(* IEC 61131-3 sources: GitHub_Test/YF_DoubleAGV/CVC_TcpTest/PLC (part 2) *)

   END_STRUCT;
END_TYPE
TYPE
    SSIO_T :
    STRUCT
        LogicalLine : DINT ;   (* Logical SSIO line.  *)
        UnitNumber : DINT ;   (* Unit id in a logical line.  *)
        InputOutputID : DINT ;   (* ID of input/output in unit.  *)
        RequestType : DINT ;   (* 0:Read input status, 1:Read output status, 2:Set output status.  *)
        SetStatus : DINT ;   (* The status to set in case of a Set output status request, 0:OFF, 1:ON, 2:Flash 1Hz.  *)
        Status : DINT ;   (* The returned status in case of a read request. Valid only when SSIO_ENO is set.  *)
        SSIO_EN : BOOL ;   (* First set SSIO address and request type then set this property to initiate a SSIO request. Clear when SSIO_ENO is set and Status has been read.  *)
        SSIO_ENO : BOOL ;   (* Set by background software when the SSIO request has been executed. For a read request this means that the reply can be read from the Status property.  *)
        Error : DINT ;   (* 0:No error, 1:Timeout.  *)

   END_STRUCT;
END_TYPE
TYPE
    CanOpenMaster_T :
    STRUCT
        MasterExecutionPeriod : DINT ;   (* Execution period for the CANopen master component. Unit is [ms].  *)
        SyncPeriod : DINT ;   (* Sync producer period given in multiples of MasterExecutionPeriod.  *)
        CollectTimeout : DINT ;   (* Collect timeout before can server enters safe state  *)
        CanMasterCmd : DINT ;   (* Command to CAN master when CanMasterEN is set, 1 = RestartCan, 2 = GoToSafeState  *)
        CanMasterCmdEN : BOOL ;   (* Commands CAN master to CanMasterCmd. Clear it when CanMasterCmdENO is set.  *)
        CanMasterCmdENO : BOOL ;   (* Set by background when commands CAN master to CanMasterCmd. Cleared when CanMasterEN is cleared.  *)
        NMTState : UDINT ;   (* The current CANopen state of the vehicle controller. Interpretation:
                        Initializing (0) = loading definition,
                        Stopped (4) = unable to start due to fatal definition error,
                        Operational (5) = The vehicle controller fully operational either in normal state or in safestate,
                        PreOperational (127) = pre-operational, configuration of slave devices,
                        Unknown (255) = state undefined, no communication with node  *)
        State : DINT ;   (* Current state of the CanOpenMaster application, 0 = NormalState, 1 = SafeState. When any error is detected that PLC does not handle, the vehicle controller will enter SafeState. Information about the error causing SafeState is available in properties StatusText, EMCY_NodeID, EMCY_Code, EMCY_ErrReg, EMCY_Byte1, etc. SafeState is a passive/diagnostic state and AllOk will be set to false.  *)
        StatusText : STRING ;   (* Text description of error that caused the vehicle controller to enter SafeState. Only valid when State = SafeState.  *)
        EMCY_BusID : DINT ;   (* Bus ID that reported the error. Only valid when State = SafeState.  *)
        EMCY_NodeID : DINT ;   (* Node ID that reported the error. Only valid when State = SafeState.  *)
        EMCY_Code : DINT ;   (* CANopen emergency code, see device documentation. Only valid when State = SafeState.  *)
        EMCY_ErrReg : DINT ;   (* Error registry. Only valid when State = SafeState.  *)
        EMCY_Byte1 : DINT ;   (* Manufacturer specific field, byte 1. Only valid when State = SafeState.  *)
        EMCY_Byte2 : DINT ;   (* Manufacturer specific field, byte 2. Only valid when State = SafeState.  *)
        EMCY_Byte3 : DINT ;   (* Manufacturer specific field, byte 3. Only valid when State = SafeState.  *)
        EMCY_Byte4 : DINT ;   (* Manufacturer specific field, byte 4. Only valid when State = SafeState.  *)
        EMCY_Byte5 : DINT ;   (* Manufacturer specific field, byte 5. Only valid when State = SafeState.  *)

   END_STRUCT;
END_TYPE
TYPE
    CanOpenEmergency_T :
    STRUCT
        EmcyEN : BOOL ;   (* Set by background when emergency data is available for a CAN device that has FailureAction set to PLC. Cleared when ENO is set.  *)
        EmcyENO : BOOL ;   (* Set by PLC when read emergency data, cleared when EN is cleared.  *)
        BusID : DINT ;   (* CAN bus id.  *)
        NodeID : DINT ;   (* CAN node id.  *)
        Code : DINT ;   (* Error code according to CANopen standard. When an emergency is generated by background program (node id is negative), the node id for the node it concerns is the last 5 bits of the code.  *)
        ErrReg : DINT ;   (* Error register according to CANopen standard.  *)
        Byte1 : DINT ;   (* Manufacturer specific error field according to CANopen standard.  *)
        Byte2 : DINT ;   (* Manufacturer specific error field according to CANopen standard.  *)
        Byte3 : DINT ;   (* Manufacturer specific error field according to CANopen standard.  *)
        Byte4 : DINT ;   (* Manufacturer specific error field according to CANopen standard.  *)
        Byte5 : DINT ;   (* Manufacturer specific error field according to CANopen standard.  *)

   END_STRUCT;
END_TYPE
TYPE
    PLCEmergency_T :
    STRUCT
        Canbus : DINT ;   (* Bus to send emergency on. 0 = first bus, 1 = second bus.  *)
        Code : DINT ;   (* Error code according to CANopen standard.  *)
        ErrReg : DINT ;   (* Error register according to CANopen standard.  *)
        Byte1 : DINT ;   (* Manufacturer specific error field according to CANopen standard.  *)
        Byte2 : DINT ;   (* Manufacturer specific error field according to CANopen standard.  *)
        Byte3 : DINT ;   (* Manufacturer specific error field according to CANopen standard.  *)
        Byte4 : DINT ;   (* Manufacturer specific error field according to CANopen standard.  *)
        Byte5 : DINT ;   (* Manufacturer specific error field according to CANopen standard.  *)
        EmcyEN : BOOL ;   (* Set by PLC when emergency data is available. Cleared by PLC when ENO is set.  *)
        EmcyENO : BOOL ;   (* Set by the vehicle controller when emergency data has been read. Cleared by the vehicle controller when EN is cleared.  *)

   END_STRUCT;
END_TYPE
TYPE
    SlavebusControl_T :
    STRUCT
        EnterPreOpEN : BOOL ;   (* Set by background when requesting to enter NMT state pre-operational. Cleared when ENO is set.  *)
        EnterPreOpENO : BOOL ;   (* Set by PLC when transition to NMT state pre-operational is granted. Cleared when EN is cleared.  *)

   END_STRUCT;
END_TYPE
TYPE
    PPA_T :
    STRUCT
        LaserScannerRef : STRING ;   (* Reference to the Laser scanner component  *)
        FrontWheelRef : STRING ;   (* Reference to the front wheel component  *)
        SteerEncRef : STRING ;   (* Symbol address where the steer encoder offset is defined. Ex: SDIO_1.SteerEncOffset  *)
        CurrentState : DINT ;   (* Current or last state of action:
0 = Idle
1 = Driving sequence 1
2 = Driving sequence 2
3 = Driving sequence 3
4 = Driving sequence 4
5 = Driving sequence 5
6 = Estimation in progress
7 = Estimation done result ok  *)
        EstimationProgress : DINT ;   (* Progressbar during calculation  *)
        CmdID : DINT ;   (* ID of current movement 1-5  *)
        ErrorID : DINT ;   (* Error Id for error condition. 0 = no error  *)
        CmdDone : DINT ;   (* Indicates completion of requested command.  *)
        SteerEncOffset : DINT ;   (* Calculated value  *)
        LaserScannerX : DINT ;   (* Calculated value  *)
        LaserScannerY : DINT ;   (* Calculated value  *)
        LaserScannerAngle : REAL ;   (* Calculated value  *)

   END_STRUCT;
END_TYPE
TYPE
    LanSerialPort_T :
    STRUCT
        Protocol : DINT ;   (* Protocol used for IP communication.  *)
        IP : STRING ;   (* In case of Protocol set to UDP client or TCP client this should be set
to the IP address of the UDP/TCP server that the PLC connects to. With
Protocol set to UDP server or TCP server this specify the IP address of
the vehicle controller which clients should use.

In the case of Protocol set to UDP server or TCP server, the special
value "LAN" means that connections are only allowed on the
LAN interface and the special value "ANY" allows connections
on both the LAN interface and the WLAN interface.

Changing the address from the PLC will result in the connection being
closed. The new IP address will be used in the next PLC loop serial
read/write.  Note! It is not possible to change the address for a
range sensor connected using a LAN-serial-adapter.  *)
        Port : DINT ;   (* In case of Protocol set to UDP client or TCP client this should be set
to the port of the UDP/TCP server that the PLC connects to. With
Protocol set to UDP server or TCP server this specify the port on the
vehicle controller that the PLC opens for connections.

Changing the port from the PLC will result in the connection being
closed. The new port will be used in the next PLC loop serial
read/write.  Note! It is not possible to change the port for a range
sensor connected using a LAN-serial-adapter.  *)
        SendBuffer : BOOL ;   (* With SendBuffer set, outgoing data is sent over IP when the PLC
function block NDC_SERIAL_WRITE is called with argument
LENGTH=0. Without SendBuffer set, data is sent immediately but each IP
packet will contain at most 32 bytes data with more IP traffic as a
result.  *)

   END_STRUCT;
END_TYPE
TYPE
    UserDefined_T :
    STRUCT
        HeartBeatTimeOut : BOOL ;   (*   *)
        MasterErrorStop : BOOL ;   (*   *)
        Boolean_3 : BOOL ;   (*   *)
        Boolean_4 : BOOL ;   (*   *)
        Boolean_5 : BOOL ;   (*   *)
        Boolean_6 : BOOL ;   (*   *)
        Boolean_7 : BOOL ;   (*   *)
        Boolean_8 : BOOL ;   (*   *)
        Boolean_9 : BOOL ;   (*   *)
        Boolean_10 : BOOL ;   (*   *)
        Boolean_11 : BOOL ;   (*   *)
        Boolean_12 : BOOL ;   (*   *)
        Boolean_13 : BOOL ;   (*   *)
        Boolean_14 : BOOL ;   (*   *)
        Boolean_15 : BOOL ;   (*   *)
        Boolean_16 : BOOL ;   (*   *)
        Boolean_17 : BOOL ;   (*   *)
        Boolean_18 : BOOL ;   (*   *)
        Boolean_19 : BOOL ;   (*   *)
        Boolean_20 : BOOL ;   (*   *)
        Boolean_21 : BOOL ;   (*   *)
        Boolean_22 : BOOL ;   (*   *)
        Boolean_23 : BOOL ;   (*   *)
        Boolean_24 : BOOL ;   (*   *)
        Boolean_25 : BOOL ;   (*   *)
        Boolean_26 : BOOL ;   (*   *)
        Boolean_27 : BOOL ;   (*   *)
        Boolean_28 : BOOL ;   (*   *)
        Boolean_29 : BOOL ;   (*   *)
        Boolean_30 : BOOL ;   (*   *)
        Integer32_1 : DINT ;   (*   *)
        Integer32_2 : DINT ;   (*   *)
        Integer32_3 : DINT ;   (*   *)
        Integer32_4 : DINT ;   (*   *)
        Integer32_5 : DINT ;   (*   *)
        Integer32_6 : DINT ;   (*   *)
        Integer32_7 : DINT ;   (*   *)
        Integer32_8 : DINT ;   (*   *)
        Integer32_9 : DINT ;   (*   *)
        Integer32_10 : DINT ;   (*   *)
        Integer32_11 : DINT ;   (*   *)
        Integer32_12 : DINT ;   (*   *)
        Integer32_13 : DINT ;   (*   *)
        Integer32_14 : DINT ;   (*   *)
        Integer32_15 : DINT ;   (*   *)
        Integer32_16 : DINT ;   (*   *)
        Integer32_17 : DINT ;   (*   *)
        Integer32_18 : DINT ;   (*   *)
        Integer32_19 : DINT ;   (*   *)
        Integer32_20 : DINT ;   (*   *)
        Integer32_21 : DINT ;   (*   *)
        TractionEncSpeed : DINT ;   (*   *)
        TractionSetSpeed : DINT ;   (*   *)
        FrontSetSpeed : DINT ;   (*   *)
        FrontEncSpeed : DINT ;   (*   *)
        FrontSetAngle : DINT ;   (*   *)
        FrontEncAngle : DINT ;   (*   *)
        RearSetSpeed : DINT ;   (*   *)
        RearEncSpeed : DINT ;   (*   *)
        RearSetAngle : DINT ;   (*   *)
        RearEncAngle : DINT ;   (*   *)
        VirFrontSetSpeed : DINT ;   (*   *)
        VirFrontEncSpeed : DINT ;   (*   *)
        VirFrontSetAngle : DINT ;   (*   *)
        VirFrontEncAngle : DINT ;   (*   *)
        VirRearSetSpeed : DINT ;   (*   *)
        VirRearEncSpeed : DINT ;   (*   *)
        VirRearSetAngle : DINT ;   (*   *)
        VirRearEncAngle : DINT ;   (*   *)
        Integer32_40 : DINT ;   (*   *)
        VirFFeedbackSpeed : DINT ;   (*   *)
        VirFFeedbackAngle : DINT ;   (*   *)
        VirRFeedbackSpeed : DINT ;   (*   *)
        VirRFeedbackAngle : DINT ;   (*   *)
        Integer32_45 : DINT ;   (*   *)
        Integer32_46 : DINT ;   (*   *)
        Integer32_47 : DINT ;   (*   *)
        Integer32_48 : DINT ;   (*   *)
        Integer32_49 : DINT ;   (*   *)
        Integer32_50 : DINT ;   (*   *)
        Integer32_51 : DINT ;   (*   *)
        Integer32_52 : DINT ;   (*   *)
        Integer32_53 : DINT ;   (*   *)
        Integer32_54 : DINT ;   (*   *)
        Integer32_55 : DINT ;   (*   *)
        Integer32_56 : DINT ;   (*   *)
        Integer32_57 : DINT ;   (*   *)
        Integer32_58 : DINT ;   (*   *)
        Integer32_59 : DINT ;   (*   *)
        Integer32_60 : DINT ;   (*   *)

   END_STRUCT;
END_TYPE
TYPE
    SDIO_T :
    STRUCT
        SteerRegP : UINT ;   (* Steering Regulator P Gain  *)
        SteerRegI : UINT ;   (* Steering Regulator I Gain  *)
        SteerRegILimit : UINT ;   (* Steering Regulator I Gain Limit  *)
        SteerRegD : UINT ;   (* Steering Regulator D Gain  *)
        SteerRegPIDLimit : UINT ;   (* Limits the effect of feedback on the steering regulator.
The unit is mV in an SDIO-FSA system.
For system only feeding the regulator output on the canbus, the value is pure binary.  *)
        SteerRegOutOffset : INT ;   (* Output offset for the steering regulator.
This offset is added to the regulator output after the PID regulation.
The unit is mV in an SDIO-FSA system.
For system only feeding the regulator output on the canbus, the value is pure binary.  *)
        SteerRegOutLimit : UINT ;   (* Total output limit of the steering regulator.
The unit is mV in an SDIO-FSA system.
For system only feeding the regulator output on the canbus, the value is pure binary.  *)
        SteerRegFailureDelay : UINT ;   (* Delay before safe state in absence of correct feedback movement  *)
        SteerRegCheckOutHysteres : UINT ;   (* Feedback movement is checked when the regulator output is larger than this level  *)
        SteerEncScale : UINT ;   (* Steering Encoder Scale  *)
        SteerEncOffset : INT ;   (* Steering Encoder Offset (Position of Sync pulse)  *)
        SteerEncSyncFilter : UINT ;   (* Steering Encoder Sync Filter Window, unit [pulses]. Filter is applied with half of the value to the right and half of the value to the left of the last valid sync pulse. 0 = Filter disabled. OBS! Disabling the sync filter can be a serious safety issue!  *)
        SteerEncSyncEmergency : BOOL ;   (* Steering Encoder Sync Emergency. 0 = Sync Emergency disabled. OBS! Disabling the sync emergency can be a serious safety issue!  *)
        SteerEncSyncEnable : BOOL ;   (* Enable signal for encoder sync mechanism. Usually needed when having a multiturning steering encoder  *)
        SyncGateInput : USINT ;   (* Digital input used for sync gate. 0 = disabled  *)
        DriveRegFeedForward : UINT ;   (* Driving Regulator FeedForward Gain  *)
        DriveRegOffset : UINT ;   (* Driving Regulator Offset  *)
        DriveRegP : UINT ;   (* Driving Regulator P Gain  *)
        DriveRegI : UINT ;   (* Driving Regulator I Gain  *)
        DriveRegILimit : UINT ;   (* Driving Regulator I Gain Limit  *)
        DriveRegD : UINT ;   (* Driving Regulator D Gain  *)
        DriveRegPIDLimit : UINT ;   (* Limits the effect of feedback on the drive regulator.
The unit is mV in an SDIO-FSA system.
For system only feeding the regulator output on the canbus, the value is pure binary.  *)
        DriveRegOutOffset : INT ;   (* Output offset for the drive regulator.
This offset is added to the regulator output after the PID regulation.
The unit is mV in an SDIO-FSA system.
For system only feeding the regulator output on the canbus, the value is pure binary.  *)
        DriveRegOutLimit : UINT ;   (* Total output limit of the drive regulator.
The unit is mV in an SDIO-FSA system.
For system only feeding the regulator output on the canbus, the value is pure binary.  *)
        DriveRegFailureDelay : UINT ;   (* Delay before safe state in absence of correct feedback movement  *)
        DriveRegCheckOutHysteres : UINT ;   (* Feedback movement is checked when the regulator output is larger than this level  *)
        DriveEncScale : UINT ;   (* Driving Encoder Scale  *)
        DigitalInput6_Polarity : BOOL ;   (* Digital Input 6 Polarity, pin #A21  *)
        FSA1Failure_Polarity : BOOL ;   (* FSA 1 Failure Polarity, pin #A20  *)
        FSA2Failure_Polarity : BOOL ;   (* FSA 2 Failure Polarity, pin #A19  *)
        DigitalInput9_Polarity : BOOL ;   (* Digital Input 9 Polarity, pin #B22  *)
        DigitalInput10_Polarity : BOOL ;   (* Digital Input 10 Polarity, pin #B23  *)
        DigitalInput11_Polarity : BOOL ;   (* Digital Input 11 Polarity, pin #A18  *)
        DigitalInput12_Polarity : BOOL ;   (* Digital Input 12 Polarity, pin #A17  *)
        DigitalOutput2_Polarity : BOOL ;   (* Digital Output 2 Polarity, pin #B7  *)
        DigitalOutput3_Polarity : BOOL ;   (* Digital Output 3 Polarity, pin #B6  *)
        DigitalOutput4_Polarity : BOOL ;   (* Digital Output 4 Polarity, pin #B5  *)
        DigitalOutput5_Polarity : BOOL ;   (* Digital Output 5 Polarity, pin #B4  *)
        DigitalOutput6_Polarity : BOOL ;   (* Digital Output 6 Polarity, pin #B1  *)
        DigitalOutput12_Polarity : BOOL ;   (* Digital Output 12 Polarity, pin #A3  *)
        AnInp1_Scale : DINT ;   (* Analog Input 1 Scale, pin #B15  *)
        AnInp2_Scale : DINT ;   (* Analog Input 2 Scale, pin #B17  *)
        AnInp3_Scale : DINT ;   (* Analog Input 3 Scale, pin #B10  *)
        AnInp4_Scale : DINT ;   (* Analog Input 4 Scale, pin #B18  *)
        AnInp5_Scale : DINT ;   (* Analog Input 5 Scale, pin #B11  *)
        AnInp6_Scale : DINT ;   (* Analog Input 6 Scale, pin #B19  *)
        AnInp7_Scale : DINT ;   (* Analog Input 7 Scale, pin #B12  *)
        AnInp8_Scale : DINT ;   (* Analog Input 8 Scale, pin #B20  *)
        AnInp9_Scale : DINT ;   (* Analog Input 9 Scale, pin #B13  *)
        AnInp10_Scale : DINT ;   (* Analog Input 10 Scale, pin #B21  *)
        AnInp11_Scale : DINT ;   (* Analog Input 11 Scale, pin #B14  *)
        AnInp1_Delta : UDINT ;   (* Asynchroneous transmission will be triggered if input has changed more than this value since last transmission.  *)
        AnInp2_Delta : UDINT ;   (* Asynchroneous transmission will be triggered if input has changed more than this value since last transmission.  *)
        AnInp3_Delta : UDINT ;   (* Asynchroneous transmission will be triggered if input has changed more than this value since last transmission.  *)
        AnInp4_Delta : UDINT ;   (* Asynchroneous transmission will be triggered if input has changed more than this value since last transmission.  *)
        AnInp5_Delta : UDINT ;   (* Asynchroneous transmission will be triggered if input has changed more than this value since last transmission.  *)
        AnInp6_Delta : UDINT ;   (* Asynchroneous transmission will be triggered if input has changed more than this value since last transmission.  *)
        AnInp7_Delta : UDINT ;   (* Asynchroneous transmission will be triggered if input has changed more than this value since last transmission.  *)
        AnInp8_Delta : UDINT ;   (* Asynchroneous transmission will be triggered if input has changed more than this value since last transmission.  *)
        AnInp9_Delta : UDINT ;   (* Asynchroneous transmission will be triggered if input has changed more than this value since last transmission.  *)
        AnInp10_Delta : UDINT ;   (* Asynchroneous transmission will be triggered if input has changed more than this value since last transmission.  *)
        AnInp11_Delta : UDINT ;   (* Asynchroneous transmission will be triggered if input has changed more than this value since last transmission.  *)
        AnInp1_Offset : DINT ;   (* Analog Input 1 Offset, pin #B15  *)
        AnInp2_Offset : DINT ;   (* Analog Input 2 Offset, pin #B17  *)
        AnInp3_Offset : DINT ;   (* Analog Input 3 Offset, pin #B10  *)
        AnInp4_Offset : DINT ;   (* Analog Input 4 Offset, pin #B18  *)
        AnInp5_Offset : DINT ;   (* Analog Input 5 Offset, pin #B11  *)
        AnInp6_Offset : DINT ;   (* Analog Input 6 Offset, pin #B19  *)
        AnInp7_Offset : DINT ;   (* Analog Input 7 Offset, pin #B12  *)
        AnInp8_Offset : DINT ;   (* Analog Input 8 Offset, pin #B20  *)
        AnInp9_Offset : DINT ;   (* Analog Input 9 Offset, pin #B13  *)
        AnInp10_Offset : DINT ;   (* Analog Input 10 Offset, pin #B21  *)
        AnInp11_Offset : DINT ;   (* Analog Input 11 Offset, pin #B14  *)
        Enc1AngularSpeed : INT ;   (* Encoder 1 Angular Speed  *)
        Enc1Angle : INT ;   (* Encoder 1 Angle  *)
        Enc1SyncValid : BOOL ;   (* Encoder 1 Sync Valid  *)
        Enc1Warning : BOOL ;   (* Encoder 1 Warning  *)
        Enc2Dist : UINT ;   (* Encoder 2 Distance  *)
        Enc2Speed : INT ;   (* Encoder 2 Speed  *)
        SetAngle : INT ;   (* Set Angle  *)
        SteerEnable : BOOL ;   (* Steering Control Enable  *)
        SetSpeed : INT ;   (* Set Speed  *)
        DriveEnable : BOOL ;   (* Driving Control Enable  *)
        Reserved_DigitalInput1 : BOOL ;   (* Reserved Digital Input 1 (Enc 1 A, pin #A14)  *)
        Reserved_DigitalInput2 : BOOL ;   (* Reserved Digital Input 2 (Enc 1 B, pin #A22)  *)
        Reserved_DigitalInput3 : BOOL ;   (* Reserved Digital Input 3 (Enc 1 Sync, pin #A7)  *)
        Reserved_DigitalInput4 : BOOL ;   (* Reserved Digital Input 4 (Enc 2 A, pin #A6)  *)
        Reserved_DigitalInput5 : BOOL ;   (* Reserved Digital Input 5 (Enc 2 B, pin #A13)  *)
        DigitalInput6 : BOOL ;   (* Digital Input 6 value, pin #A21  *)
        FSA1Failure : BOOL ;   (* FSA 1 Failure value, pin #A20  *)
        FSA2Failure : BOOL ;   (* FSA 2 Failure value, pin #A19  *)
        DigitalInput9 : BOOL ;   (* Digital Input 9 value, pin #B22  *)
        DigitalInput10 : BOOL ;   (* Digital Input 10 value, pin #B23  *)
        DigitalInput11 : BOOL ;   (* Digital Input 11 value, pin #A18  *)
        DigitalInput12 : BOOL ;   (* Digital Input 12 value, pin #A17  *)
        AllOK_DigitalOutput1 : BOOL ;   (* Reserved Digital Output 1 (All-OK, pin #B8)  *)
        DigitalOutput2 : BOOL ;   (* Digital Output 2 value, pin #B7  *)
        DigitalOutput3 : BOOL ;   (* Digital Output 3 value, pin #B6  *)
        DigitalOutput4 : BOOL ;   (* Digital Output 4 value, pin #B5  *)
        DigitalOutput5 : BOOL ;   (* Digital Output 5 value, pin #B4  *)
        DigitalOutput6 : BOOL ;   (* Digital Output 6 value, pin #B1  *)
        DigitalOutput12 : BOOL ;   (* Digital Output 12 value, pin #A3  *)
        AnalogInput1 : INT ;   (* Analog Input 1 value, pin #B15. The value is the applied input voltage (in Volts) * Scale + Offset  *)
        AnalogInput2 : INT ;   (* Analog Input 2 value, pin #B17. The value is the applied input voltage (in Volts) * Scale + Offset  *)
        AnalogInput3 : INT ;   (* Analog Input 3 value, pin #B10. The value is the applied input voltage (in Volts) * Scale + Offset  *)
        AnalogInput4 : INT ;   (* Analog Input 4 value, pin #B18. The value is the applied input voltage (in Volts) * Scale + Offset  *)
        AnalogInput5 : INT ;   (* Analog Input 5 value, pin #B11. The value is the applied input voltage (in Volts) * Scale + Offset  *)
        AnalogInput6 : INT ;   (* Analog Input 6 value, pin #B19. The value is the applied input voltage (in Volts) * Scale + Offset  *)
        AnalogInput7 : INT ;   (* Analog Input 7 value, pin #B12. The value is the applied input voltage (in Volts) * Scale + Offset  *)
        AnalogInput8 : INT ;   (* Analog Input 8 value, pin #B20. The value is the applied input voltage (in Volts) * Scale + Offset  *)
        AnalogInput9 : INT ;   (* Analog Input 9 value, pin #B13. The value is the applied input voltage (in Volts) * Scale + Offset  *)
        AnalogInput10 : INT ;   (* Analog Input 10 value, pin #B21. The value is the applied input voltage (in Volts) * Scale + Offset  *)
        AnalogInput11 : INT ;   (* Analog Input 11 value, pin #B14. The value is the applied input voltage (in Volts) * Scale + Offset  *)
        PWMOutput1 : INT ;   (* PWM Output 1 value, pin #A5. The value is the duty cycle of the output.  *)
        PWMOutput2 : INT ;   (* PWM Output 2 value, pin #A12. The value is the duty cycle of the output.  *)
        PWMOutput3 : INT ;   (* PWM Output 3 value, pin #A11. The value is the duty cycle of the output.  *)
        Reg1Output : INT ;   (* Regulator 1 output value  *)
        Reg2Output : INT ;   (* Regulator 2 output value  *)
        GroundFaultEvent : BOOL ;   (* If set to true, a ground fault will cause a system event 229.  *)
        GroundFaultActive : BOOL ;   (* True if a ground fault is present  *)
        Temperature : DINT ;   (* Current temperature  *)
        XV_Out : DINT ;   (* Current xv out voltage  *)
        B_Plus : DINT ;   (* Current b plus voltage  *)
        BusID : DINT ;   (* CAN bus ID  *)
        NodeID : DINT ;   (* CAN node ID  *)
        FailureAction : DINT ;   (* 0 = Background, the background programs takes action when an error occur in the device. 1 = PLC, no action from background program. The error should be handled by the PLC application.  *)
        ActiveInSafeState : BOOL ;   (* Decides if the device will start up in safe state.  *)
        NMTState : UDINT ;   (* The current CANopen state of the device.  *)
        SdoBufferSize : DINT ;   (* The current size of the client SDO buffer (read/write SDO's from the vehicle controller to this device).  *)

   END_STRUCT;
END_TYPE

TYPE
    NDC8_T :
    STRUCT
	NavInit : NavInit_T;
	    Mcd : MCD7P_T;
	    Position : Position_T;
	    Guidance : Guidance_T;
	    Autoinsert : Autoinsert_T;
	    Opt : GenericDisplay_T;
	    LayoutPosition : LayoutPosition_T;
	    Automatic : Automatic_T;
	    Manual : Manual_T;
	    BlackBox : BlackBox_T;
	    LocalOrder : LocalOrder_T;
	    SSIO : SSIO_T;
	    SegmentTrigger : SegmentTrigger_T;
	    PointTrigger : PointTrigger_T;
	    LoadDocking : LoadDocking_T;
	    LoadOperation : LoadOperation_T;
	    CANBus1 : CANBus_T;
	    CANBus2 : CANBus_T;
	    VehicleControl : VehicleControl_T;
	    VehicleOptions : VehicleOptions_T;
	    PLC_Application : PLC_Application_T;
	    COM1 : SerialPort_RS232_T;
	    COM2 : SerialPort_RS422_T;
	    COM3 : SerialPort_RS485_T;
	    Master : Master_T;
	    Vmc : Vmc_T;
	    Wlan : Wlan_T;
	    OMPLC : OMPLC_T;
	    VehicleApplication : VehicleApplication_T;
	    Layout : Layout_T;
	    CanOpenMaster : CanOpenMaster_T;
	    CanOpenEmergency : CanOpenEmergency_T;
	    PLCEmergency : PLCEmergency_T;
	    SlavebusControl : SlavebusControl_T;
	    UserDefined : UserDefined_T;
	    ExternalPath : ExternalPath_T;
	    BlockedInfo : BlockedInfo_T;
	    FrontWheel : WheelSD_T;
	    LS2000 : LS2000Scanner_T;
	    COM5 : LanSerialPort_T;
	    Vehicle : Vehicle_T;
	    PPA : PPA_T;
	    TurnSignal : TurnSignal_T;
	    LaserNavigator : LaserNavigator_T;
	    ReflectorInit : ReflectorInit_T;
	    NaturalNavigator : NaturalNavigator_T;
	    VehicleNavigator : VehicleNavigator_T;
	    SDIO : SDIO_T;

   END_STRUCT;
END_TYPE

(* ---- ClientReceiveData_FB.ST ---- *)
FUNCTION_BLOCK ClientReceiveData_FB
VAR_EXTERNAL
NDC8 : NDC8_T;
END_VAR

VAR_INPUT

END_VAR

VAR_OUTPUT

END_VAR

VAR
serial_read  : NDC8_SERIAL_READ;
TcpPort_CRC : TcpPort_CRC_FB;
MasterVehicleID : dint;
MasterTravelDir : dint;
MasterTractionEncSpeed : dint;
MasterPositionX : dint;
MasterPositionY : dint;
MasterDistOpPoint : dint;
MasterOpCode : dint;
ClientDistOpPoint : dint;
DevDist: dint;
SpeedScale : real;
TestValue: dint;
Count,CountValue : dint;
SpeedTemp : dint;
PreMasterPositionX : dint;
MasterRemainDis : dint;
PreDevDist : dint;
P_Scale,D_Scale : real;
MasterFlag : dint;
PreMasterPositionY : dint;
MasterAngle : dint;
IdevDist : dint;
I_Scale : real;
PI : real;
PP : real;
VirX : dint;
PP_DINT,PI_DINT : dint;
Flag : bool;
OverCount : dint;
Icount : dint;
ClientRemainDis : dint;
PreClientPositionX : dint;
PreClientPositionY : dint;
DevPercent,P_DevPercent_Scale,PP_DevPercent : real;
DevRemainDis : dint;
PP_Curve,P_Curve_Scale,PI_Curve,I_Curve_Scale : real;
PP_Curve_DINT,PI_Curve_DINT : dint;
CalSetAddSpeed : dint;
MasterTractionSetSpeed : dint;
ShouldRemainDis : dint;
PreMasterRemainDis,PreClientRemainDis : dint;
TxtValue : real;
PreDevRemainDis,DdevDist,PD_Curve_DINT : dint;
PD_Curve,D_Curve_Scale : real;

PreHeartBeatClient : dint;
NoHeartBeat : bool;
HeartBeatTimeOut : ton;
ClientX,DevX,PreDevX,V1,T2,ClientY,DevY,DevAngle : dint;
T1,HuDu : REAL;

SendData : Array[1..32] of Byte;
tempHigh_X,tempHigh_Y,tempHigh_MX,tempHigh_MY,tempHigh_CX,tempHigh_CY : dint;
serial_write  : NDC8_SERIAL_WRITE;
FlagCount : dint;
AngleScale : real;
MasterAngle2 : dint;
VV1 : real;
END_VAR

serial_read(Port:='COM5');

TcpPort_CRC(cBuffer:=serial_read.Data,CrcLength:=28);

if serial_read.Data[1]=16#4A and serial_read.Data[2]=16#54
	and serial_read.Data[29]=TcpPort_CRC.CrcLow and serial_read.Data[30]=TcpPort_CRC.CrcHigh then

	MasterVehicleID := byte_to_dint(serial_read.Data[3]);

	MasterTravelDir := byte_to_dint(serial_read.Data[4]);

	MasterTractionEncSpeed := byte_to_dint(serial_read.Data[5])*256 + byte_to_dint(serial_read.Data[6]) ;

	MasterPositionX := byte_to_dint(serial_read.Data[7])*167777216 + byte_to_dint(serial_read.Data[8])*65536
						+ byte_to_dint(serial_read.Data[9])*256 + byte_to_dint(serial_read.Data[10]) + VirX;

	MasterPositionY := byte_to_dint(serial_read.Data[11])*167777216 + byte_to_dint(serial_read.Data[12])*65536
						+ byte_to_dint(serial_read.Data[13])*256 + byte_to_dint(serial_read.Data[14]) ;

	MasterDistOpPoint := byte_to_dint(serial_read.Data[15])*256 + byte_to_dint(serial_read.Data[16]) ;

	MasterOpCode  := byte_to_dint(serial_read.Data[17]);

	MasterRemainDis := byte_to_dint(serial_read.Data[18])*256 + byte_to_dint(serial_read.Data[19]) ;

	MasterFlag := byte_to_dint(serial_read.Data[20]);

	MasterTractionSetSpeed := byte_to_dint(serial_read.Data[21])*256 + byte_to_dint(serial_read.Data[22]) ;

	HeartBeatClient := byte_to_dint(serial_read.Data[23]);

	AErrorStop := byte_to_bool(serial_read.Data[24]);

	MasterAngle := byte_to_dint(serial_read.Data[25])*256 + byte_to_dint(serial_read.Data[26]) ;

	MasterAngle2 := byte_to_dint(serial_read.Data[27])*256 + byte_to_dint(serial_read.Data[28]) ;
end_if;

(*if NDC8.OMPLC.Data91=1 and MasterFlag=1 then
	if HeartBeatClient=1 then
		HeartBeatMaster := 0;
	elsif HeartBeatClient=0 then
		HeartBeatMaster := 1;
	end_if;

	PreHeartBeatClient := HeartBeatClient;

	NoHeartBeat := (PreHeartBeatClient=HeartBeatClient);
	HeartBeatTimeOut(IN:=NoHeartBeat,PT:=t#1s);
	StopHeartBeatTimeOut := HeartBeatTimeOut.Q;
end_if;*)

if NDC8.OMPLC.Data91=1 and MasterFlag=1 then

	if NDC8.SegmentTrigger.LeftTurn or NDC8.SegmentTrigger.RightTurn then
		FlagCount := 1;

		if dint_to_real(MasterAngle2)/100.0>=(180.0-VV1) and dint_to_real(MasterAngle2)/100.0<=(180.0+VV1) then
			AngleScale := (9496.0/5752.0 - 1.0)/VV1 * abs(abs((dint_to_real(MasterAngle2)/100.0-180.0))-VV1);
		elsif dint_to_real(MasterAngle2)/100.0>=(270.0-VV1) and dint_to_real(MasterAngle2)/100.0<=(270.0+VV1) then
			AngleScale := (9496.0/5752.0 - 1.0)/VV1 * abs(abs((dint_to_real(MasterAngle2)/100.0-270.0))-VV1);
		else
			AngleScale := 0.0;
		end_if;

		SetAddSpeed := real_to_dint(dint_to_real(MasterTractionSetSpeed)*9496.0/5752.0/(1.0+AngleScale));

		ClientX := real_to_dint(sin(dint_to_real(MasterAngle)*3.14159/180.0)*2367.0) + MasterPositionX;

		if MasterAngle>=90 and MasterAngle<=270 and NDC8.VehicleControl.TravelDir=1 then
			DevX := NDC8.Position.X - ClientX;
		elsif MasterAngle>=90 and MasterAngle<=270 and NDC8.VehicleControl.TravelDir=0 then
			DevX := ClientX - NDC8.Position.X;
		elsif (MasterAngle<90 or MasterAngle>270) and NDC8.VehicleControl.TravelDir=1 then
			DevX := ClientX - NDC8.Position.X;
		elsif (MasterAngle<90 or MasterAngle>270) and NDC8.VehicleControl.TravelDir=0 then
			DevX := NDC8.Position.X - ClientX;
		end_if;

(* --------------------------------PID Adjustment------------------------------------------------- *)
		(* P Adjust *)
		P_Curve_Scale := 0.65;
		PP_Curve := P_Curve_Scale * dint_to_real(DevX);
		if PP_Curve<-150.0 then
			PP_Curve := -150.0;
		elsif PP_Curve>150.0 then
			PP_Curve := 150.0;
		end_if;
		(* I Adjust *)
		if (abs(DevX) > 30)  or Icount > 10 then
			IdevDist := 0;
			Icount := 0;
		else
			IdevDist := DevX + IdevDist;
			Icount := Icount + 1;
		end_if;
		I_Curve_Scale := 0.1;
  		PI_Curve := I_Curve_Scale*dint_to_real(IdevDist);
		if PI_Curve<-20.0 then
			PI_Curve := -20.0;
		elsif PI_Curve>20.0 then
			PI_Curve := 20.0;
		end_if;

		(* D Adjust *)
		if abs(DevX) < 20 then
			DdevDist := DdevDist + DevX - PreDevX ;
		else
			DdevDist := 0;
		end_if;
		PreDevX := DevX;
		PD_Curve := D_Curve_Scale*dint_to_real(DdevDist);
(* --------------------------------PID Adjustment------------------------------------------------- *)

		SetAddSpeed := SetAddSpeed + real_to_dint(PP_Curve+PI_Curve+PD_Curve) ;
		SetAddSpeed := MIN(NDC8.Vehicle.MaxSpeed,SetAddSpeed);

		SendData[1] := 16#4A;
		SendData[2] := 16#54;
		tempHigh_X := NDC8.Position.X / 65536;
		SendData[3] := word_to_byte(SHR(dint_to_word(tempHigh_X),8));
		SendData[4] := dint_to_byte(tempHigh_X);
		SendData[5] := word_to_byte(SHR(dint_to_word(NDC8.Position.X),8));
		SendData[6] := dint_to_byte(NDC8.Position.X);

		tempHigh_Y := NDC8.Position.Y / 65536;
		SendData[7] := word_to_byte(SHR(dint_to_word(tempHigh_Y),8));
		SendData[8] := dint_to_byte(tempHigh_Y);
		SendData[9] := word_to_byte(SHR(dint_to_word(NDC8.Position.Y),8));
		SendData[10] := dint_to_byte(NDC8.Position.Y);

		tempHigh_MX := MasterPositionX / 65536;
		SendData[11] := word_to_byte(SHR(dint_to_word(tempHigh_MX),8));
		SendData[12] := dint_to_byte(tempHigh_MX);
		SendData[13] := word_to_byte(SHR(dint_to_word(MasterPositionX),8));
		SendData[14] := dint_to_byte(MasterPositionX);

		tempHigh_MY := MasterPositionY / 65536;
		SendData[15] := word_to_byte(SHR(dint_to_word(tempHigh_MY),8));
		SendData[16] := dint_to_byte(tempHigh_MY);
		SendData[17] := word_to_byte(SHR(dint_to_word(MasterPositionY),8));
		SendData[18] := dint_to_byte(MasterPositionY);

		tempHigh_CX := ClientX / 65536;
		SendData[19] := word_to_byte(SHR(dint_to_word(tempHigh_CX),8));
		SendData[20] := dint_to_byte(tempHigh_CX);
		SendData[21] := word_to_byte(SHR(dint_to_word(ClientX),8));
		SendData[22] := dint_to_byte(ClientX);

	(*	tempHigh_CY := ClientY / 65536;
		SendData[23] := word_to_byte(SHR(dint_to_word(tempHigh_CY),8));
		SendData[24] := dint_to_byte(tempHigh_CY);
		SendData[25] := word_to_byte(SHR(dint_to_word(ClientY),8));
		SendData[26] := dint_to_byte(ClientY);			*)
		SendData[23] := word_to_byte(SHR(dint_to_word(MasterAngle),8));
		SendData[24] := dint_to_byte(MasterAngle);
		SendData[25] := word_to_byte(SHR(dint_to_word(NDC8.Position.Angle),8));
		SendData[26] := dint_to_byte(NDC8.Position.Angle);

		SendData[27] := word_to_byte(SHR(dint_to_word(DevX),8));
		SendData[28] := dint_to_byte(DevX);

		SendData[29] := word_to_byte(SHR(dint_to_word(SetAddSpeed),8));
		SendData[30] := dint_to_byte(SetAddSpeed);

		serial_write( port:='COM5',data:=SendData,length:=30 );

	(*	a:= TRACE_DINT('DevX',DevX);
		a:= TRACE_DINT('ClientX',ClientX);
		a:= TRACE_DINT('ClientY',ClientY);
		a:= TRACE_DINT('NDC8.Position.X',NDC8.Position.X);
		a:= TRACE_DINT('NDC8.Position.Y',NDC8.Position.Y);
		a:= TRACE_DINT('NDC8.Position.Angle',NDC8.Position.Angle);
		a:= TRACE_DINT('MasterPositionX',MasterPositionX);
		a:= TRACE_DINT('MasterPositionY',MasterPositionY);
		a:= TRACE_DINT('MasterAngle',MasterAngle);
		a:= TRACE_DINT('ClientRemainDis',NDC8.LayoutPosition.RemainingDistance);
		a:= TRACE_DINT('MasterRemainDis',MasterRemainDis);
		a:= TRACE_DINT('DevRemainDis',DevRemainDis);
		a:= TRACE_DINT('ShouldRemainDis',ShouldRemainDis);
		a:= TRACE_DINT('PP_Curve_DINT',PP_Curve_DINT);
		a:= TRACE_DINT('PI_Curve_DINT',PI_Curve_DINT);
		a:= TRACE_DINT('SetAddSpeed',SetAddSpeed);
		a:= TRACE_DINT('CalSetAddSpeed',CalSetAddSpeed);
		a:= TRACE_DINT('MasterTractionSetSpeed',MasterTractionSetSpeed);
		a:= TRACE_DINT('MasterTractionEncSpeed',MasterTractionEncSpeed);
		a:= TRACE_DINT('ClientEncSpeed',NDC8.UserDefined.TractionEncSpeed);
		a:= TRACE_DINT('ClientSetSpeed',NDC8.UserDefined.TractionSetSpeed);*)
	else

(*	if NDC8.SegmentTrigger.GateOpen then
		if MasterPositionY=PreMasterPositionY then
			;
		else
	 		DevDist := NDC8.Position.Y - MasterPositionY + 4367;
			PreMasterPositionY := MasterPositionY;
		end_if;
	else
		if MasterPositionX=PreMasterPositionX then
			;
		else
	 		DevDist := NDC8.Position.X - MasterPositionX;
			PreMasterPositionX := MasterPositionX;
		end_if;
	end_if;*)

		if NDC8.SegmentTrigger.GateOpen then
			FlagCount := 2;
			if MasterPositionY=PreMasterPositionY then
				;
			else
				if (NDC8.Position.Y-PreClientPositionY)<=0 and (MasterPositionY-PreMasterPositionY)<0 then
			 		DevDist := NDC8.Position.Y - MasterPositionY;
				elsif (NDC8.Position.Y-PreClientPositionY)>=0 and (MasterPositionY-PreMasterPositionY)>0 then
					DevDist := MasterPositionY - NDC8.Position.Y;
				end_if;

				if not Flag then
					Flag := true;
				else
					if abs(DevDist-PreDevDist) > 10 then
						if OverCount > 0 then
							;
						else
					  		DevDist := PreDevDist;
					   	    OverCount := OverCount + 1;
						end_if;
					else
						OverCount := 0;
					end_if;
				end_if;
				PreMasterPositionY := MasterPositionY;
				PreClientPositionY := NDC8.Position.Y;
			end_if;

		else
			FlagCount := 3;
			if MasterPositionX=PreMasterPositionX then
				;
			else
				if (NDC8.Position.X-PreClientPositionX)<=0 and (MasterPositionX-PreMasterPositionX)<0 then
			 		DevDist := NDC8.Position.X - MasterPositionX;
				elsif (NDC8.Position.X-PreClientPositionX)>=0 and (MasterPositionX-PreMasterPositionX)>0 then
					DevDist := MasterPositionX - NDC8.Position.X;
				end_if;

				if not Flag then
					Flag := true;
				else
					if abs(DevDist-PreDevDist) > 10 then
						if OverCount > 0 then
							;
						else
						   DevDist := PreDevDist;
						   OverCount := OverCount + 1;
						end_if;
					else
						OverCount := 0;
					end_if;
				end_if;

				PreMasterPositionX := MasterPositionX;
				PreClientPositionX := NDC8.Position.X;
			end_if;
	end_if;

(*	a:= TRACE_DINT('OverCount',OverCount);
	a:= TRACE_DINT('PreDevDist',PreDevDist);
	a:= TRACE_DINT('DevDist',DevDist);
	a:= TRACE_DINT('NDC8.Position.X',NDC8.Position.X);
	a:= TRACE_DINT('MasterPositionX',MasterPositionX);
	a:= TRACE_DINT('NDC8.Position.Y',NDC8.Position.Y);
	a:= TRACE_DINT('MasterPositionY',MasterPositionY);	*)

	PreDevDist := DevDist;

(* --------------------------------PID Adjustment------------------------------------------------- *)
	(* P Adjust *)
	P_Scale := 0.55;
	PP := P_Scale*dint_to_real(DevDist);
	if PP<-150.0 then
		PP := -150.0;
	elsif PP>150.0 then
		PP := 150.0;
	end_if;
	(* I Adjust *)
	if abs(DevDist) > 10 or Icount > 10 then
		IdevDist := 0;
		Icount := 0;
	else
		IdevDist := DevDist + IdevDist;
		Icount := Icount + 1;
	end_if;
	I_Scale := 0.1;
	PI := I_Scale*dint_to_real(IdevDist);
	if PI<-10.0 then
		PI := -10.0;
	elsif PI>10.0 then
		PI := 10.0;
	end_if;
(* --------------------------------PID Adjustment------------------------------------------------- *)

	SetAddSpeed := real_to_dint(PP + PI) ;

(*	PP_DINT := real_to_dint(PP);
	PI_DINT := real_to_dint(PI);
	a:= TRACE_DINT('PP',PP_DINT);
	a:= TRACE_DINT('PI',PI_DINT);*)
(*	SetAddSpeed := real_to_dint(P_Scale*dint_to_real(DevDist) + D_Scale*dint_to_real(DevDist - PreDevDist) );*)
(*	SetAddSpeed := real_to_dint(P_Scale*dint_to_real(DevDist) + D_Scale*dint_to_real(DevDist - PreDevDist)  + PI  );*)

(*	SetAddSpeed := MasterTractionEncSpeed + real_to_dint(P_Scale*dint_to_real(DevDist) + D_Scale*dint_to_real(DevDist - PreDevDist) );*)

(*	a:= TRACE_DINT('MasterTractionEncSpeed',MasterTractionEncSpeed);
	a:= TRACE_DINT('ClientEncSpeed',NDC8.UserDefined.TractionEncSpeed);
	a:= TRACE_DINT('SetAddSpeed',SetAddSpeed);*)

	end_if;
else
	Flag := false;
	Icount := 0;
	OverCount := 0;
	PreDevDist := 0;
	DevDist := 0;
	DevRemainDis := 0;
	SetAddSpeed := 0;
end_if;

END_FUNCTION_BLOCK

(* ---- GoGroup_FB.ST ---- *)
FUNCTION_BLOCK GoGroup_FB
VAR_EXTERNAL
NDC8 : NDC8_T;
END_VAR

VAR_INPUT

END_VAR

VAR_OUTPUT

END_VAR

VAR
 NAVINIT : NAVINIT_FB;
 LocalOrder : LocalOrder_FB;
 GroupRtrig : r_trig;
 MasterOnPoint : bool;
 ClientOnPoint : bool;
 state : dint;
 MasterFlag : bool;
 ClientFlag : bool;
END_VAR
(*
GroupRtrig(CLK:=NDC8.UserDefined.Boolean_25);

if GoGroup then

case state of
0:
	if NDC8.Vehicle.VehicleID=2 then
		state := 1;
		MasterFlag := false;
	end_if;
	if NDC8.Vehicle.VehicleID=3 then
		ClientFlag := false;
		state := 2;
	end_if;

1:
	if NDC8.Vehicle.VehicleID=2 and NDC8.LayoutPosition.InSystem and NDC8.VehicleControl.OperationMode=0 and NDC8.LayoutPosition.Point<>1
		and not MasterFlag then
		NDC8.LocalOrder.DestPoint:=1;
		NDC8.LocalOrder.OpCode:=0;
		LocalOrder();
		if LocalOrder.Finished then
			MasterOnPoint := true;
			MasterFlag := true;
			state := 3;
		end_if;
	elsif NDC8.Vehicle.VehicleID=2 and NDC8.LayoutPosition.InSystem and NDC8.VehicleControl.OperationMode=0 and NDC8.LayoutPosition.Point=1 then
		MasterOnPoint := true;
		state := 3;
	end_if;

2:
	if NDC8.Vehicle.VehicleID=3 and NDC8.LayoutPosition.InSystem and NDC8.VehicleControl.OperationMode=0 and NDC8.LayoutPosition.Point<>3
		and not ClientFlag then
		NDC8.LocalOrder.DestPoint:=3;
		NDC8.LocalOrder.OpCode:=0;
		LocalOrder();
		if LocalOrder.Finished then
			ClientOnPoint := true;
			ClientFlag := true;
		end_if;
	end_if;

end_case;
end_if;
*)

;
END_FUNCTION_BLOCK

(* ---- SMControl_FB.ST ---- *)
FUNCTION_BLOCK SMControl_FB
VAR_EXTERNAL
NDC8 : NDC8_T;
END_VAR

VAR_INPUT

END_VAR

VAR_OUTPUT

END_VAR

VAR

END_VAR

if NDC8.OMPLC.Data1=1 then
	NDC8.UserDefined.Boolean_25 := true;
	if NDC8.Vehicle.VehicleID=2 then
		if TCP_OK and MasterOnInitOK then
			NDC8.OMPLC.Data3 := 1;
		else
			NDC8.OMPLC.Data3 := 0;
		end_if;
	elsif NDC8.Vehicle.VehicleID=3 then
		if TCP_OK then
			NDC8.OMPLC.Data3 := 1;
		else
			NDC8.OMPLC.Data3 := 0;
		end_if;
	end_if;
elsif NDC8.OMPLC.Data1=2 then
	NDC8.UserDefined.Boolean_25 := false;
	if NDC8.Vehicle.VehicleID=2 then
		if not NDC8.UserDefined.Boolean_25 and MasterOffInitOK then
			NDC8.OMPLC.Data3 := 1;
		else
			NDC8.OMPLC.Data3 := 0;
		end_if;
	elsif NDC8.Vehicle.VehicleID=3 then
		if not TCP_OK and ClientOffInitOK then
			NDC8.OMPLC.Data3 := 1;
		else
			NDC8.OMPLC.Data3 := 0;
		end_if;
	end_if;
end_if;

END_FUNCTION_BLOCK

(* ---- TCP_DriverTrasfer_FB.ST ---- *)
FUNCTION_BLOCK TCP_DriverTrasfer_FB
VAR_EXTERNAL
NDC8 : NDC8_T;
DriverSend_ValueByte:ARRAY[1..500] OF Byte;
DriverReceive_ValueByte:ARRAY[1..500] OF Byte;
END_VAR

VAR_INPUT

END_VAR

VAR_OUTPUT

END_VAR

VAR
serial_read : NDC8_SERIAL_READ;
serial_write : NDC8_SERIAL_WRITE;
StartDelayTon : TON;
StartDelay : BOOL;
init : BOOL;
TcpPortState : DINT;
ConvWord:WORD;			(*Sum of the two first bytes*)
ConvByteL:int;			(*Low byte*)
ConvByteH:int;			(*High byte*)
start_adress : int;
num_words : dint;
X: INT;
Y: INT;
Z: INT;
Index:DINT;
SendLength : int;
Function_Code : dint;
StartWriteTON : ton;
StartWrite : bool;
TcpPort_CRC : TcpPort_CRC_FB;
ReadData : ARRAY[1..32] OF BYTE;
ReadLength : int;
crclow : int;
crchigh : int;
CheckLength : uint;
initite : bool;
WriteData : Array[1..32] of Byte;
count : dint;

VirDriverSendData : VirDriverSendData_FB;
VirDriverReceiveData : VirDriverReceiveData_FB;
END_VAR

StartDelayTon(IN:=StartDelay,PT:=t#100ms);
StartWriteTON(IN:=StartWrite,PT:=t#50ms);

if not NDC8.UserDefined.Boolean_25 then
	TcpPortState := 0;
	TCP_OK := false;
end_if;

(* Always read COM7 to check if some information from Host *)
(*serial_read(port := 'COM7');*)

if not Init then
	serial_write.port := 'COM7';
	serial_read.port := 'COM7';
(*	serial_write.port := 'COM8';
	serial_read.port := 'COM8';*)
	Init := true;
end_if;

case TcpPortState of
0:
(*	StartDelay := true;
	if StartDelayTon.Q then
	TcpPortState := 50;
	StartDelay := false;
	end_if;*)
	TcpPortState := 50;

50:
	if NDC8.Vehicle.VehicleID=2 then
		TcpPortState := 1;
	elsif NDC8.Vehicle.VehicleID=3 then
		TcpPortState := 2;
	end_if;

1:
	WriteData[1] := 16#4A;
	WriteData[2] := 16#54;
	WriteData[3] := 16#03; (* Virtual Vehicle ID *)
	WriteData[4] := 16#03; (* Function Code *)
	VirDriverSendData();   (* Vir Vehicle speed and angle , data[5] to data[12] *)
	if VirDriverSendData.Finish then
		Y := 5;
		X := 5;
		For Index:=1 to 6 By 1 Do
			WriteData[Y] := DriverSend_ValueByte[X];
			Y:=Y+1;
			X:=X+1;
			WriteData[Y] := DriverSend_ValueByte[X];
			Y:=Y+1;
			X:=X+1;
		end_for;
		CheckLength := 16;
		crclow := 17;
		crchigh := 18;
		TcpPort_CRC(cBuffer:=WriteData,CrcLength:=CheckLength);
		WriteData[crclow]:=TcpPort_CRC.CrcLow;
		WriteData[crchigh]:=TcpPort_CRC.CrcHigh;
		SendLength := 18;
		StartWrite := true;
		TcpPortState := 80;
	end_if;

80:
	(*serial_write(port := 'COM7');
	serial_write.length := dint_to_int(SendLength);*)
	if NDC8.UserDefined.Boolean_25 then
		if StartWriteTON.Q then
			serial_write( port:='COM7',data:=WriteData,length:=SendLength );
			serial_write( port:='COM7',data:=WriteData,length:=0 );
			StartWrite := false;
			TcpPortState:=2;
		else
			TcpPortState:=2;
		end_if;
	else
		TcpPortState:=0;
	end_if;
(*	if serial_write.sent<>0 then
		TcpPortState:=2;
	end_if;	*)

2:
	serial_read(port := 'COM7');
	(* check data valid?is it matchs the vehicle? *)
	ReadLength := serial_read.length;
	ReadData := serial_read.data;
	if ReadLength >0 and ReadData[1]=16#4A and ReadData[2]=16#54
		and (NDC8.Vehicle.VehicleID = byte_to_dint(ReadData[3])) then
		if (byte_to_dint(ReadData[3])=3 or byte_to_dint(ReadData[3])=2) then
		TCP_OK := true;
		Count := 0;
		TcpPortState := 3;
		else
		Count := 0;
		TcpPortState := 3;
		end_if;
	else
		Count := Count + 1;
		if Count>10 or not NDC8.UserDefined.Boolean_25 then
			TCP_OK := false;
			Count := 0;
		end_if;
		TcpPortState := 0;
	end_if;
(*
30:
	serial_read(port := 'COM7');
	ReadLength := serial_read.length;
	ReadData := serial_read.data;
	if ReadLength >0 and ReadData[1]=16#4A and ReadData[2]=16#54
		and (NDC8.Vehicle.VehicleID = byte_to_dint(ReadData[3])) then
		TcpPortState := 3;
		TCP_OK := true;
	else
		TcpPortState := 0;
		TCP_OK := false;
	end_if;
*)
3:
	(* check the data read from Tcp Port is right or not *)
	crclow := ReadLength - 1;
	crchigh := ReadLength;
	CheckLength := int_to_uint(ReadLength - 2);
	TcpPort_CRC(cBuffer:=ReadData,CrcLength:=CheckLength);
	if ReadData[crclow]=TcpPort_CRC.CrcLow and ReadData[crchigh]=TcpPort_CRC.CrcHigh then
		TcpPortState := 4;
	else
		TcpPortState := 0;
	end_if;

4:
	Function_Code := byte_to_dint(ReadData[4]);
	case Function_Code of
	3:
	(*	ISD_ValueByte_Read();
		if ISD_ValueByte_Read.finish then
		TcpPortState := 10;
		end_if;*)
		TcpPortState := 11;
   16:
  		TcpPortState := 20;
end_case;

20:
	(* reveive vie vehicle speed and angle *)
	Y := 5;
	X := 5;
	For Index:=1 to 6 By 1 Do
	DriverReceive_ValueByte[Y] := ReadData[X];
	Y:=Y+1;
	X:=X+1;
	DriverReceive_ValueByte[Y] := ReadData[X];
	Y:=Y+1;
	X:=X+1;
	end_for;
	VirDriverReceiveData();
	if VirDriverReceiveData.Finish then
		TcpPortState := 0;
	end_if;

11:
	Y := 5;
	X := 5;
	For Index:=1 to 6 By 1 Do
	DriverReceive_ValueByte[Y] := ReadData[X];
	Y:=Y+1;
	X:=X+1;
	DriverReceive_ValueByte[Y] := ReadData[X];
	Y:=Y+1;
	X:=X+1;
	end_for;
	VirDriverReceiveData();
	if VirDriverReceiveData.Finish then
		TcpPortState := 12;
	end_if;

12:
	WriteData[1] := 16#4A;
	WriteData[2] := 16#54;
	WriteData[3] := 16#02; (* Master Vehicle ID *)
	WriteData[4] := 16#10; (* Function Code, Virtual Vehicle return data to Master Vehicle *)
	VirDriverSendData();   (* Vir Vehicle speed and angle , data[5] to data[12] *)
	if VirDriverSendData.Finish then
		Y := 5;
		X := 5;
		For Index:=1 to 6 By 1 Do
			WriteData[Y] := DriverSend_ValueByte[X];
			Y:=Y+1;
			X:=X+1;
			WriteData[Y] := DriverSend_ValueByte[X];
			Y:=Y+1;
			X:=X+1;
		end_for;
		CheckLength := 16;
		crclow := 17;
		crchigh := 18;
		TcpPort_CRC(cBuffer:=WriteData,CrcLength:=CheckLength);
		WriteData[crclow]:=TcpPort_CRC.CrcLow;
		WriteData[crchigh]:=TcpPort_CRC.CrcHigh;
		SendLength := 18;
		StartWrite := true;
		TcpPortState := 81;
	end_if;

81:
	(*serial_write(port := 'COM7');
	serial_write.length := dint_to_int(SendLength);*)
	if StartWriteTON.Q then
		serial_write( port:='COM7',data:=WriteData,length:=SendLength );
		serial_write( port:='COM7',data:=WriteData,length:=0 );
		StartWrite := false;
		TcpPortState:=0;
	end_if;
(*	if serial_write.sent<>0 then
		TcpPortState:=0;
	end_if;*)

end_case;

END_FUNCTION_BLOCK

(* ---- VirDriverReceiveData_FB.ST ---- *)
FUNCTION_BLOCK VirDriverReceiveData_FB
VAR_EXTERNAL
NDC8 : NDC8_T;
DriverReceive_ValueByte:ARRAY[1..500] OF Byte;
END_VAR

VAR_INPUT

END_VAR

VAR_OUTPUT
Finish : bool;
END_VAR

VAR
HighDint : dint;
LowDint : dint;
END_VAR
if NDC8.Vehicle.VehicleID=2 then (* Master Vehicle *)
	HighDint := byte_to_dint(DriverReceive_ValueByte[5]);
	LowDint  := byte_to_dint(DriverReceive_ValueByte[6]);
	if DriverReceive_ValueByte[13]=1 then
		NDC8.UserDefined.VirFrontEncSpeed := (HighDint*256 + LowDint) - NDC8.UserDefined.VirFFeedbackSpeed;
	else
		NDC8.UserDefined.VirFrontEncSpeed := -(HighDint*256 + LowDint) - NDC8.UserDefined.VirFFeedbackSpeed;
	end_if;

	HighDint := byte_to_dint(DriverReceive_ValueByte[7]);
	LowDint  := byte_to_dint(DriverReceive_ValueByte[8]);
	if DriverReceive_ValueByte[14]=1 then
		NDC8.UserDefined.VirFrontEncAngle := -(HighDint*256 + LowDint) - NDC8.UserDefined.VirFFeedbackAngle;
	else
		NDC8.UserDefined.VirFrontEncAngle := HighDint*256 + LowDint - NDC8.UserDefined.VirFFeedbackAngle;
	end_if;

	HighDint := byte_to_dint(DriverReceive_ValueByte[9]);
	LowDint  := byte_to_dint(DriverReceive_ValueByte[10]);
	if DriverReceive_ValueByte[15]=1 then
		NDC8.UserDefined.VirRearEncSpeed := HighDint*256 + LowDint - NDC8.UserDefined.VirRFeedbackSpeed;
	else
		NDC8.UserDefined.VirRearEncSpeed := -(HighDint*256 + LowDint) - NDC8.UserDefined.VirRFeedbackSpeed;
	end_if;

	HighDint := byte_to_dint(DriverReceive_ValueByte[11]);
	LowDint  := byte_to_dint(DriverReceive_ValueByte[12]);
	if DriverReceive_ValueByte[16]=1 then
		NDC8.UserDefined.VirRearEncAngle := -(HighDint*256 + LowDint) - NDC8.UserDefined.VirRFeedbackAngle;
	else
		NDC8.UserDefined.VirRearEncAngle := HighDint*256 + LowDint - NDC8.UserDefined.VirRFeedbackAngle;
	end_if;

elsif NDC8.Vehicle.VehicleID=3 then  (* Client Vehicle *)
	HighDint := byte_to_dint(DriverReceive_ValueByte[5]);
	LowDint  := byte_to_dint(DriverReceive_ValueByte[6]);
	if DriverReceive_ValueByte[13]=1 then
		NDC8.UserDefined.FrontSetSpeed := HighDint*256 + LowDint;
	else
		NDC8.UserDefined.FrontSetSpeed := -(HighDint*256 + LowDint);
	end_if;

	HighDint := byte_to_dint(DriverReceive_ValueByte[7]);
	LowDint  := byte_to_dint(DriverReceive_ValueByte[8]);
	if DriverReceive_ValueByte[14]=1 then
		NDC8.UserDefined.FrontSetAngle := -(HighDint*256 + LowDint);
	else
		NDC8.UserDefined.FrontSetAngle := HighDint*256 + LowDint;
	end_if;

	HighDint := byte_to_dint(DriverReceive_ValueByte[9]);
	LowDint  := byte_to_dint(DriverReceive_ValueByte[10]);
	if DriverReceive_ValueByte[15]=1 then
		NDC8.UserDefined.RearSetSpeed := HighDint*256 + LowDint;
	else
		NDC8.UserDefined.RearSetSpeed := -(HighDint*256 + LowDint);
	end_if;

	HighDint := byte_to_dint(DriverReceive_ValueByte[11]);
	LowDint  := byte_to_dint(DriverReceive_ValueByte[12]);
	if DriverReceive_ValueByte[16]=1 then
		NDC8.UserDefined.RearSetAngle := -(HighDint*256 + LowDint);
	else
		NDC8.UserDefined.RearSetAngle := HighDint*256 + LowDint;
	end_if;
end_if;

Finish := true;

END_FUNCTION_BLOCK

(* ---- VirDriverSendData_FB.ST ---- *)
FUNCTION_BLOCK VirDriverSendData_FB
VAR_EXTERNAL
NDC8 : NDC8_T;
DriverSend_ValueByte:ARRAY[1..500] OF Byte;
END_VAR

VAR_INPUT

END_VAR

VAR_OUTPUT
Finish : bool;
END_VAR

VAR
HighDint : dint;
LowDint : dint;
END_VAR

if NDC8.Vehicle.VehicleID= 2 then (* Master Vehicle *)
	HighDint := abs(NDC8.UserDefined.VirFrontSetSpeed)/256;
	LowDint :=  abs(NDC8.UserDefined.VirFrontSetSpeed) - (HighDint*256);
	DriverSend_ValueByte[5] := dint_to_byte(HighDint);
	DriverSend_ValueByte[6] := dint_to_byte(LowDint);

	HighDint := abs(NDC8.UserDefined.VirFrontSetAngle)/256;
	LowDint :=  abs(NDC8.UserDefined.VirFrontSetAngle) - (HighDint*256);
	DriverSend_ValueByte[7] := dint_to_byte(HighDint);
	DriverSend_ValueByte[8] := dint_to_byte(LowDint);

	HighDint := abs(NDC8.UserDefined.VirRearSetSpeed)/256;
	LowDint :=  abs(NDC8.UserDefined.VirRearSetSpeed) - (HighDint*256);
	DriverSend_ValueByte[9] := dint_to_byte(HighDint);
	DriverSend_ValueByte[10] := dint_to_byte(LowDint);

	HighDint := abs(NDC8.UserDefined.VirRearSetAngle)/256;
	LowDint :=  abs(NDC8.UserDefined.VirRearSetAngle) - (HighDint*256);
	DriverSend_ValueByte[11] := dint_to_byte(HighDint);
	DriverSend_ValueByte[12] := dint_to_byte(LowDint);

	if NDC8.UserDefined.VirFrontSetSpeed<0 then
		DriverSend_ValueByte[13] := 1;
	else
		DriverSend_ValueByte[13] := 0;
	end_if;
	if NDC8.UserDefined.VirFrontSetAngle<0 then
		DriverSend_ValueByte[14] := 1;
	else
		DriverSend_ValueByte[14] := 0;
	end_if;
	if NDC8.UserDefined.VirRearSetSpeed<0 then
		DriverSend_ValueByte[15] := 1;
	else
		DriverSend_ValueByte[15] := 0;
	end_if;
	if NDC8.UserDefined.VirRearSetAngle<0 then
		DriverSend_ValueByte[16] := 1;
	else
		DriverSend_ValueByte[16] := 0;
	end_if;

elsif NDC8.Vehicle.VehicleID= 3 then (* Client Vehicle *)
	HighDint := abs(NDC8.UserDefined.FrontEncSpeed)/256;
	LowDint :=  abs(NDC8.UserDefined.FrontEncSpeed) - (HighDint*256);
	DriverSend_ValueByte[5] := dint_to_byte(HighDint);
	DriverSend_ValueByte[6] := dint_to_byte(LowDint);

	HighDint := abs(NDC8.UserDefined.FrontEncAngle)/256;
	LowDint :=  abs(NDC8.UserDefined.FrontEncAngle) - (HighDint*256);
	DriverSend_ValueByte[7] := dint_to_byte(HighDint);
	DriverSend_ValueByte[8] := dint_to_byte(LowDint);

	HighDint := abs(NDC8.UserDefined.RearEncSpeed)/256;
	LowDint :=  abs(NDC8.UserDefined.RearEncSpeed) - (HighDint*256);
	DriverSend_ValueByte[9] := dint_to_byte(HighDint);
	DriverSend_ValueByte[10] := dint_to_byte(LowDint);

	HighDint := abs(NDC8.UserDefined.RearEncAngle)/256;
	LowDint :=  abs(NDC8.UserDefined.RearEncAngle) - (HighDint*256);
	DriverSend_ValueByte[11] := dint_to_byte(HighDint);
	DriverSend_ValueByte[12] := dint_to_byte(LowDint);

	if NDC8.UserDefined.FrontEncSpeed<0 then
		DriverSend_ValueByte[13] := 1;
	else
		DriverSend_ValueByte[13] := 0;
	end_if;
	if NDC8.UserDefined.FrontEncAngle<0 then
		DriverSend_ValueByte[14] := 1;
	else
		DriverSend_ValueByte[14] := 0;
	end_if;
	if NDC8.UserDefined.RearEncSpeed<0 then
		DriverSend_ValueByte[15] := 1;
	else
		DriverSend_ValueByte[15] := 0;
	end_if;
	if NDC8.UserDefined.RearEncAngle<0 then
		DriverSend_ValueByte[16] := 1;
	else
		DriverSend_ValueByte[16] := 0;
	end_if;

end_if;

	Finish := true;

END_FUNCTION_BLOCK

(* ---- VirWheelControl_FB.ST ---- *)
FUNCTION_BLOCK VirWheelControl_FB
VAR_EXTERNAL
NDC8 : NDC8_T;
END_VAR

VAR_INPUT

END_VAR

VAR_OUTPUT

END_VAR

VAR
TCP_DriverTrasfer : TCP_DriverTrasfer_FB;
END_VAR

if NDC8.UserDefined.Boolean_25 then
	TCP_DriverTrasfer();
	if NDC8.Vehicle.VehicleID=3 then
		NDC8.VehicleControl.PlcSelect := 1;
		NDC8.VehicleControl.PlcSelectMask := 15;
		NDC8.VehicleControl.PlcSetSteerEnable := 1;
		NDC8.VehicleControl.PlcSetDriveEnable := 1;

		NDC8.LS2000.NavActive := 0;
	(*	NDC8.Manual.PlcSelect := 1;
		NDC8.Manual.PlcSelectMask := 4;
		NDC8.Manual.PlcSetOperationMode := 1;*)
	(*	if NDC8.UserDefined.FrontSetAngle>11500 then
			NDC8.UserDefined.FrontSetAngle := NDC8.UserDefined.FrontSetAngle - 65792;
		end_if;
		if NDC8.UserDefined.RearSetAngle>11500 then
			NDC8.UserDefined.RearSetAngle := NDC8.UserDefined.RearSetAngle - 65792;
		end_if;
		if NDC8.UserDefined.FrontSetSpeed>1500 then
			NDC8.UserDefined.FrontSetSpeed := NDC8.UserDefined.FrontSetSpeed - 65792;
		end_if;
		if NDC8.UserDefined.RearSetSpeed>1500 then
			NDC8.UserDefined.RearSetSpeed := NDC8.UserDefined.RearSetSpeed - 65792;
		end_if;*)
		if TCP_OK then
			NDC8.FrontWheel.PlcSetSpeed := NDC8.UserDefined.FrontSetSpeed;
			NDC8.FrontWheel.PlcSetAngle := NDC8.UserDefined.FrontSetAngle;
			NDC8.RearWheel.PlcSetSpeed  := NDC8.UserDefined.RearSetSpeed;
			NDC8.RearWheel.PlcSetAngle  := NDC8.UserDefined.RearSetAngle;
		else
			NDC8.FrontWheel.PlcSetSpeed := 0;
			NDC8.RearWheel.PlcSetSpeed  := 0;
		end_if;
	end_if;
else
	NDC8.VehicleControl.PlcSelect := 0;
	NDC8.VehicleControl.PlcSelectMask := 0;
	NDC8.VehicleControl.PlcSetSteerEnable := 0;
	NDC8.VehicleControl.PlcSetDriveEnable := 0;

(*	NDC8.Manual.PlcSelect := 1;
	NDC8.Manual.PlcSelectMask := 4;
	NDC8.Manual.PlcSetOperationMode := 1;*)
	NDC8.LS2000.NavActive := 1;

	NDC8.UserDefined.VirFrontEncSpeed := NDC8.UserDefined.VirFrontSetSpeed - NDC8.UserDefined.VirFFeedbackSpeed;
	NDC8.UserDefined.VirFrontEncAngle := NDC8.UserDefined.VirFrontSetAngle - NDC8.UserDefined.VirFFeedbackAngle;
	NDC8.UserDefined.VirRearEncSpeed  := NDC8.UserDefined.VirRearSetSpeed - NDC8.UserDefined.VirRFeedbackSpeed;
	NDC8.UserDefined.VirRearEncAngle  := NDC8.UserDefined.VirRearSetAngle - NDC8.UserDefined.VirRFeedbackAngle;
end_if;

END_FUNCTION_BLOCK

(* ---- WheelXYControl_FB.ST ---- *)
FUNCTION_BLOCK WheelXYControl_FB
VAR_EXTERNAL
NDC8 : NDC8_T;
END_VAR

VAR_INPUT

END_VAR

VAR_OUTPUT

END_VAR

VAR

END_VAR

if NDC8.UserDefined.Boolean_25 then
	if NDC8.Vehicle.VehicleID=2 then
		NDC8.FrontWheel.X := 1590;
		NDC8.FrontWheel.Y := 300;
		NDC8.RearWheel.X := 810;
		NDC8.RearWheel.Y := 300;
		NDC8.VirFrontWheel.X := -1590;
		NDC8.VirFrontWheel.Y := -300;
		NDC8.VirRearWheel.X := -810;
		NDC8.VirRearWheel.Y := -300;
		NDC8.LS2000.X := 1860;
	end_if;
else
	NDC8.FrontWheel.X := 390;
	NDC8.FrontWheel.Y := 300;
	NDC8.RearWheel.X := -390;
	NDC8.RearWheel.Y := 300;
	NDC8.VirFrontWheel.X := -1590;
	NDC8.VirFrontWheel.Y := -300;
	NDC8.VirRearWheel.X := -810;
	NDC8.VirRearWheel.Y := -300;
	NDC8.LS2000.X := 660;
end_if;

END_FUNCTION_BLOCK

(* ---- ReplaceMe.ST ---- *)
PROGRAM ReplaceMe
VAR_EXTERNAL
NDC8 : NDC8_T;
END_VAR

VAR_GLOBAL
END_VAR

VAR
TcpPortSend : TcpPortSend_FB;
TcpPortReceive : TcpPortReceive_FB;
END_VAR

if NDC8.CanOpenMaster.NMTState=5 and NDC8.CanOpenMaster.State=0 then
	TcpPortReceive();
	TcpPortSend();
end_if;
END_PROGRAM
